(* PLC project circuit_braker, Dassault Systèmes ControlBuild 2024x *)
(* stored: creationDateTime 2023-10-03T11:13:23-01:00 *)

(* This module simulates a circuit braker. The trip results in a power outage. *)
FUNCTION_BLOCK equipment_library.circuit_braker
  VAR_INPUT
    energyBefore : BOOL := true;
    sensorSupply : BOOL := true;
  END_VAR
  VAR_OUTPUT
    thermal : BOOL := false;
    energyAfter : BOOL := false;
  END_VAR
  VAR CONSTANT
    wiringLogic : BOOL := false;
  END_VAR
  VAR
    d_electric : BOOL := false;
    v_d_electric : BOOL := false;
  END_VAR


ACTION C_source_code:
/* ----------------------------------------------------------------	*/
/* Type : Model of Operative Behaviour					*/
/* Category :  Power								*/
/* Author : Dassault Systemes						*/
/* Update date : June 2018							*/
/* ----------------------------------------------------------------	*/
/* This module simulates a circuit braker.				*/
/* The trip results in a power outage.					*/
/* It returns its state.							*/
/* ----------------------------------------------------------------	*/

/* ----------------------------------------------------------------	*/
/* Management of feedback to Control Part					*/
/*     if a fault is required, the thermal circuit braker 		*/
/*		 takes a preset state.					*/
/*	if there is no power supply for sensor 				*/
/*         thermal contactor returns nothing				*/
/*     else thermal contactor returns its state combined with		*/
/*	    wiring logic (its default value is : negative).		*/
/* ----------------------------------------------------------------	*/

if (d_electric) thermal=v_d_electric;
else
	if (sensorSupply) thermal= sensorSupply ^ !wiringLogic;
	else thermal=0;

/* ----------------------------------------------------------------	*/
/* Management of the energy flow						*/
/*     Energy passes through the circuit braker				*/
/* if there is no electric fault.						*/
/* ----------------------------------------------------------------	*/
energyAfter = energyBefore & ! d_electric;
END_ACTION
END_FUNCTION_BLOCK
